// TIA Portal V18 export
DATA_BLOCK "Dest_DB"   // DB4
{ S7_Optimized_Access := 'FALSE' }
   VAR
      IN1 : Array[0..5] of Int;
      IN2 : Int;
      IN3 : Int;
      IN4 : Int;
   END_VAR
BEGIN
END_DATA_BLOCK
